# EPICS substitutions: galil/3-6/GalilTestApp/Db/galil_userdef_records.substitutions
# P - PV prefix
# PORT - asyn port
# ADDR 0 - 63
# EPICSNAME - PV suffix
# P:EPICSNAME_MONITOR
# P:EPICSNAME_STATUS
# P:EPICSNAME_SP
# P:EPICSNAME_CMD

# GALILSTR - is a galil command or variable
# eg. TI0, SB 1, user variable name, etc

# DRVCMD = VAR (GALILSTR is a galil variable)
# DRVCMD = CMD (GALILSTR is a galil command)
# ADDR 0 - 63.  VAR and CMD are separately numbered from 0 - 63

# SCAN = use I/O Intr when EPICS only will change the value.
#        use Periodic scan when external will change value.
# PINI = YES will push autosave or default value to controller at startup

file "$(GALIL)/GalilSup/Db/galil_userdef_records.template"
{
    pattern
    {P,        M,   PORT,    ADDR, PREC, SCAN,      MTRTYPE, MTRON, EGU  }
    {"DMC01:", "A", "Galil", 0,    3,   "Passive",  "3",     "0",   "mm" }
}
